Staubli VAL3: JointStateMsg.pjx

--- JointStateMsg.pjx ---
Parameters version=s7.7.2 stackSize=5000 millimeterUnit=true
Program file=start.pgx
Program file=stop.pgx
Data file=JointStateMsg.dtx
Type name=Body path=Disk://ros_libs/Body/Body.pjx
Type name=Prefix path=Disk://ros_libs/Prefix/Prefix.pjx
Type name=Header path=Disk://ros_libs/Header/Header.pjx
Type name=JointState path=Disk://ros_libs/JointState/JointState.pjx

--- JointStateMsg.dtx ---
public Header header
  [0]
    num nMsgType
    num nCommType
    num nReplyCode
    num nData[12]
public Body body
  [0]
    num nData[44]
public JointState jointState
  [0]
    num nSeq
    num nJoints[10]
public Prefix prefix
  [0]
    num nLength
    num nData[4]
